{attribute 'qualified_only'}
//{attribute 'strict'}
TYPE eCurrentState :
(
	OFF := 0,
	STANDBY := 1,
	MANUAL := 2,
	AVG_PWR_CTR := 3,
	INST_PWR_CTR := 4
) INT;
END_TYPE

(* stored: Version 1.1.0.1, ProductVersion 3.1.4024.2
   DUT eCurrentState: Id {700a5dfc-da19-47b6-aafd-fb15c4a39634} *)
